PROGRAM FUN_GetPublicIp

VAR_INPUT
	ParamNetID				: STRING :='' ; // Unit ID of the PC with internet connexion
	IN_CmdStart 			: BOOL;
	IN_DirExe				: STRING;
END_VAR
VAR_OUTPUT
	OUT_Completed			: BOOL;
END_VAR

VAR
	RS_Start				: RS;
	TRIG_Completed			: R_TRIG;
	TRIG_Start				: R_TRIG;
	start_process			: NT_StartProcess;
END_VAR


TRIG_Start(ClK := IN_CmdStart);
TRIG_Completed(CLK := OUT_Completed);


RS_Start(SET := TRIG_Start.Q, RESET1 := TRIG_Completed.Q);

IF RS_Start.Q1 THEN
	IN_CmdStart := FALSE;
	start_process
	(
		NETID := ParamNetID,
		PATHSTR := Concat(IN_DirExe, 'GetPublicIp.exe'),
		DIRNAME := IN_DirExe,
		COMNDLINE := '',
		Start := TRUE
	);
ELSE
	start_process(START := FALSE);
END_IF

IF TRIG_Completed.Q THEN
	OUT_Completed := FALSE;
END_IF

END_PROGRAM

(* stored: Version 1.1.0.1, ProductVersion 3.1.4024.6
   POU FUN_GetPublicIp: Id {97220610-ae82-49a6-8b44-e52a9a53d05e}, SpecialFunc None *)
